TYPE ST_PNInput_ParallelOperation :
STRUCT
	Controlbits			:	DWORD;
	//b_DetectSlaves	
	r_ActivePower		:	DWORD;
	r_reactivePower		:	DWORD;
END_STRUCT
END_TYPE

(* stored: Version 1.1.0.1, ProductVersion 3.1.4024.12
   DUT ST_PNInput_ParallelOperation: Id {64bc7339-2efa-47ed-9e96-ac2dbe321ebf} *)
